TYPE ST_Machine_HMI EXTENDS ST_HmiFunction :
	STRUCT
		Override : LREAL := 100.0;
	END_STRUCT
END_TYPE

(* stored: Version 1.1.0.1, ProductVersion 3.1.4026.18
   DUT ST_Machine_HMI: Id {c9be57c9-2b6c-4078-bf80-004ccab94b9d} *)
